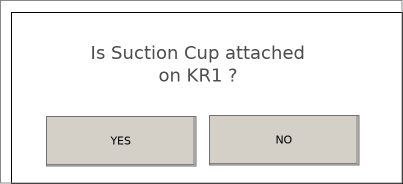
VISUALIZATION MSG_EOAT_SUCTION  // 403x184
    RoundedRectangle (11,12 392x172)
    Button (46,116 150x50), "YES"
        OnMouseClick: execute { GVL.KR1_EOAT_FILL:= FALSE; GVL.KR1_EOAT_SUCTION:= TRUE; }
        OnMouseClick: CloseDialog Dialog=MSG_EOAT_SUCTION, Result=Yes, NumpadKeypadSet=True
    Button (209,115 150x50), "NO"
        OnMouseClick: execute { GVL.KR1_EOAT_SUCTION:= FALSE; }
        OnMouseClick: CloseDialog Dialog=MSG_EOAT_SUCTION, Result=No, NumpadKeypadSet=True
    Label (80,20 236x88), "Is Suction Cup attached on KR1 ?"
END_VISUALIZATION

(* stored: Version 1.1.0.1, ProductVersion 3.1.4024.12
   Visu MSG_EOAT_SUCTION: Id {83d7d187-99cf-4a33-891d-9b074f0b217f} *)
